FUNCTION_BLOCK CncHFunctions
VAR_INPUT
	nFuncNr				: UDINT;		(* Number of H-function *)
	nArg				: DINT;		(* Argument of H-Function *)
END_VAR
VAR
	argument52 :DINT :=0;
	argument522 :DINT :=0;
END_VAR
VAR_OUTPUT
	Busy :BOOL;
END_VAR

(* ========================================================= *)
(*    FUN: CncHFunctions                                     *)
(* --------------------------------------------------------- *)
(*   Desc:                                                   *)
(* Author: JRM                                               *)
(*   Date: 20.12.2017                                        *)
(*   Rev.: 1.0                                               *)
(* ========================================================= *)
Busy:= TRUE;

CASE nFuncNr OF
	53:
		CASE nArg OF
			0: IOs.IO_Out_Vent_Quadro1:=FALSE;
				IOs.IO_Out_Vent_Quadro2:=FALSE;
				
			1: IOs.IO_Out_Vent_Quadro1:=TRUE;
				IOs.IO_Out_Vent_Quadro2:=FALSE;
				
			2: IOs.IO_Out_Vent_Quadro1:=TRUE;
				IOs.IO_Out_Vent_Quadro2:=TRUE;
		END_CASE
		Busy:=FALSE;
	

		
END_CASE

END_FUNCTION_BLOCK

(* stored: Version 1.1.0.1, ProductVersion 3.1.4020.12
   POU CncHFunctions: Id {ab541539-e7bf-42bd-8ae8-1d87f6d822e1}, SpecialFunc None *)
